// TIA Portal V20 export
DATA_BLOCK "LBP_SentronPac"   // DB1001
TITLE = SENTRON PAC
{ S7_Optimized_Access := 'FALSE'; DB_Accessible_From_OPC_UA := 'FALSE' }
AUTHOR : SINUMERIK
FAMILY : SINUMERIK_ONE
VERSION : 6.24
// Interface between user program and operating software, contains signals for SENTRON PAC energy monitoring devices / Interface entre programme utilisateur et logiciel d'exploitation, contient des signaux pour unités de surveillance de l'énergie SENTRON PAC
// stored: AutoNumber false, DBAccessibleFromOPCUA false, DBAccessibleFromWebserver false
   VAR RETAIN
      ManualVal { ExternalWritable := 'False'} : Bool;   // Display of manual value / Affichage de la valeur manuelle
      SentronPacMach { ExternalWritable := 'False'} : Bool;   // Sentron PAC represented machine / Machine représentée par Sentron PAC
      FeedInEnergyReadSP { ExternalWritable := 'False'} : Bool;   // Feed-in energy read from Sentron PAC / Énergie alimentée mesurée par Sentron PAC
      FeedBackEnergyReadSP { ExternalWritable := 'False'} : Bool;   // Feed back energy read from Sentron PAC / Énergie réinjectée mesurée par Sentron PAC
      FeedInEnergyReadAuxil { ExternalWritable := 'False'} : Bool;   // Feed-in energy read auxiliary / Énergie alimentée, mesurée par AUX
      FeedBackEnergyReadAuxil { ExternalWritable := 'False'} : Bool;   // Feed back energy read auxiliary / Énergie réinjectée, mesurée par AUX
      res0_6 { ExternalWritable := 'False'} : Bool;   // Reserved / Réservé
      res0_7 { ExternalWritable := 'False'} : Bool;   // Reserved / Réservé
      MeasAuto { ExternalWritable := 'False'} : Bool;   // Measurement by PLC basic program / Mesure par programme de base AP
      res1_1 { ExternalWritable := 'False'} : Bool;   // Reserved / Réservé
      res1_2 { ExternalWritable := 'False'} : Bool;   // Reserved / Réservé
      res1_3 { ExternalWritable := 'False'} : Bool;   // Reserved / Réservé
      res1_4 { ExternalWritable := 'False'} : Bool;   // Reserved / Réservé
      res1_5 { ExternalWritable := 'False'} : Bool;   // Reserved / Réservé
      res1_6 { ExternalWritable := 'False'} : Bool;   // Reserved / Réservé
      res1_7 { ExternalWritable := 'False'} : Bool;   // Reserved / Réservé
      MeasAct : Bool;   // HMI -> PLC: Active measurement / IHM->AP : Mesure active
      res2_1 { ExternalWritable := 'False'} : Bool;   // Reserved / Réservé
      res2_2 { ExternalWritable := 'False'} : Bool;   // Reserved / Réservé
      res2_3 { ExternalWritable := 'False'} : Bool;   // Reserved / Réservé
      res2_4 { ExternalWritable := 'False'} : Bool;   // Reserved / Réservé
      res2_5 { ExternalWritable := 'False'} : Bool;   // Reserved / Réservé
      res2_6 { ExternalWritable := 'False'} : Bool;   // Reserved / Réservé
      res2_7 { ExternalWritable := 'False'} : Bool;   // Reserved / Réservé
      EStateOn { ExternalWritable := 'False'} : Bool;   // Energy state on / État énergie activé
      res3_1 { ExternalWritable := 'False'} : Bool;   // Reserved / Réservé
      res3_2 { ExternalWritable := 'False'} : Bool;   // Reserved / Réservé
      res3_3 { ExternalWritable := 'False'} : Bool;   // Reserved / Réservé
      res3_4 { ExternalWritable := 'False'} : Bool;   // Reserved / Réservé
      res3_5 { ExternalWritable := 'False'} : Bool;   // Reserved / Réservé
      res3_6 { ExternalWritable := 'False'} : Bool;   // Reserved / Réservé
      res3_7 { ExternalWritable := 'False'} : Bool;   // Reserved / Réservé
      ManualValue { ExternalWritable := 'False'} : Real;   // Manual value / Valeur manuelle
      ActivePowerItem { ExternalWritable := 'False'} : Real;   // Active power item / Puissance active position
      ActiveEnergyItem { ExternalWritable := 'False'} : Real;   // Active energy item / Énergie active position
      ReactiveEnergyItem { ExternalWritable := 'False'} : Real;   // Reactive energy item / Énergie réactive position
      ActivePowerSentron { ExternalWritable := 'False'} : Real;   // Active power from Sentron / Puissance active par Sentron
      ActiveEnergySentron { ExternalWritable := 'False'} : Real;   // Active energy from Sentron / Énergie active par Sentron
      ReactiveEnergySentron { ExternalWritable := 'False'} : Real;   // Reactive energy from Sentron / Énergie réactive par Sentron
      ActiveEnergyDay { ExternalWritable := 'False'} : Real;   // Active energy day / Énergie active jour
      ReactiveEnergyDay { ExternalWritable := 'False'} : Real;   // Reactive energy day / Énergie réactive jour
      ActiveEnergyPrevDay { ExternalWritable := 'False'} : Real;   // Active energy previous day / Énergie active jour précédent
      ReactiveEnergyPrevDay { ExternalWritable := 'False'} : Real;   // Reactive energy previous day / Énergie réactive jour précédent
      ActiveEnergyMonth { ExternalWritable := 'False'} : Real;   // Active energy month / Énergie active mois
      ReactiveEnergyMonth { ExternalWritable := 'False'} : Real;   // Reactive energy month / Énergie réactive mois
      ActiveEnergyPrevMonth { ExternalWritable := 'False'} : Real;   // Active energy previous month / Énergie active mois précédent
      ReactiveEnergyPrevMonth { ExternalWritable := 'False'} : Real;   // Reactive energy previous month / Énergie réactive mois précédent
      ActiveEnergyYear { ExternalWritable := 'False'} : Real;   // Active energy year / Énergie active année
      ReactiveEnergyYear { ExternalWritable := 'False'} : Real;   // Reactive energy year / Énergie réactive année
      ActiveEnergyPrevYear { ExternalWritable := 'False'} : Real;   // Active energy previous year / Énergie active année précédente
      ReactiveEnergyPrevYear { ExternalWritable := 'False'} : Real;   // Reactive energy previous year / Énergie réactive année précédente
      res80 { ExternalWritable := 'False'} : Byte;   // Reserved / Réservé
      res81 { ExternalWritable := 'False'} : Byte;   // Reserved / Réservé
      res82 { ExternalWritable := 'False'} : Byte;   // Reserved / Réservé
      res83 { ExternalWritable := 'False'} : Byte;   // Reserved / Réservé
      res84 { ExternalWritable := 'False'} : Byte;   // Reserved / Réservé
      res85 { ExternalWritable := 'False'} : Byte;   // Reserved / Réservé
      res86 { ExternalWritable := 'False'} : Byte;   // Reserved / Réservé
      res87 { ExternalWritable := 'False'} : Byte;   // Reserved / Réservé
      res88 { ExternalWritable := 'False'} : Real;   // Reserved / Réservé
      res92 { ExternalWritable := 'False'} : Real;   // Reserved / Réservé
      ProductionAct { ExternalWritable := 'False'} : Byte;
      ErrDBD20_NAN { ExternalWritable := 'False'} : Bool;   // DBD20: invalid (not a number) / DBD20 : non valide (pas un nombre)
      ErrDBD24_NAN { ExternalWritable := 'False'} : Bool;   // DBD24: invalid (not a number) / DBD24 : non valide (pas un nombre)
      ErrDBD28_NAN { ExternalWritable := 'False'} : Bool;   // DBD28: invalid (not a number) / DBD28 : non valide (pas un nombre)
      res97_3 { ExternalWritable := 'False'} : Bool;   // Reserved / Réservé
      res97_4 { ExternalWritable := 'False'} : Bool;   // Reserved / Réservé
      res97_5 { ExternalWritable := 'False'} : Bool;   // Reserved / Réservé
      res97_6 { ExternalWritable := 'False'} : Bool;   // Reserved / Réservé
      res97_7 { ExternalWritable := 'False'} : Bool;   // Reserved / Réservé
      ErrDBD104_NAN { ExternalWritable := 'False'} : Bool;   // DBD104: invalid (not a number) / DBD104 : non valide (pas un nombre)
      ErrDBD144_NAN { ExternalWritable := 'False'} : Bool;   // DBD144: invalid (not a number) / DBD144 : non valide (pas un nombre)
      ErrDBD184_NAN { ExternalWritable := 'False'} : Bool;   // DBD184: invalid (not a number) / DBD184 : non valide (pas un nombre)
      ErrDBD224_NAN { ExternalWritable := 'False'} : Bool;   // DBD224: invalid (not a number) / DBD224 : non valide (pas un nombre)
      ErrDBD264_NAN { ExternalWritable := 'False'} : Bool;   // DBD264: invalid (not a number) / DBD264 : non valide (pas un nombre)
      ErrDBD304_NAN { ExternalWritable := 'False'} : Bool;   // DBD304: invalid (not a number) / DBD304 : non valide (pas un nombre)
      ErrDBD344_NAN { ExternalWritable := 'False'} : Bool;   // DBD344: invalid (not a number) / DBD344 : non valide (pas un nombre)
      ErrDBD384_NAN { ExternalWritable := 'False'} : Bool;   // DBD384: invalid (not a number) / DBD384 : non valide (pas un nombre)
      ErrDBD424_NAN { ExternalWritable := 'False'} : Bool;   // DBD424: invalid (not a number) / DBD424 : non valide (pas un nombre)
      ErrDBD464_NAN { ExternalWritable := 'False'} : Bool;   // DBD464: invalid (not a number) / DBD464 : non valide (pas un nombre)
      res99_2 { ExternalWritable := 'False'} : Bool;   // Reserved / Réservé
      res99_3 { ExternalWritable := 'False'} : Bool;   // Reserved / Réservé
      res99_4 { ExternalWritable := 'False'} : Bool;   // Reserved / Réservé
      res99_5 { ExternalWritable := 'False'} : Bool;   // Reserved / Réservé
      res99_6 { ExternalWritable := 'False'} : Bool;   // Reserved / Réservé
      res99_7 { ExternalWritable := 'False'} : Bool;   // Reserved / Réservé
      CtrlE_AuxDevice { ExternalWritable := 'False'} : Array[1..10] of Struct
         ProcessAux : Bool;   // Auxiliary present and to be processed / AUX présent et prêt au traitement
         ReadEnergy : Bool;   // Actual values are refreshed; bit is auto-reset / Les valeurs réelles sont actualisées ; le bit est réinitialisé automatiquement
         MeasAct : Bool;   // Measurement values are computed / Calcul des valeurs de mesure en cours
         MeasMode : Bool;   // Difference of actual values is stored / La différence des valeurs réelles est enregistrée
         InputMode : Bool;   // INPUT "ActivePowerAux" is energy in kWh / INPUT "ActivePowerAux" représente l'énergie en kWh
         res0_5 : Bool;
         res0_6 : Bool;
         ResetAux : Bool;   // Auxiliary data are deleted / Les données AUX sont supprimées
         res1 : Byte;   // Reserved / Réservé
         res2 : Word;   // Reserved / Réservé
         ActivePowerAux : Real;   // [kW]/[kWh] power/energy of auxiliary, written by customer / [kW]/[kWh] puissance/énergie AUX, renseignée par le client
         ActiveEnAux : Real;   // [kWh] actual value of fed-in-energy / [kWh] valeur réelle de l'énergie consommée
         ReActiveEnAux : Real;   // [kWh] actual value of fed-back energy / [kWh] valeur réelle de l'énergie réinjectée
         ActiveEnAuxMeasON : Real;   // [kWh] value of fed-in-energy at start of measurement / [kWh] valeur réelle de l'énergie consommée au début de la mesure
         ReActiveEnAuxMeasON : Real;   // [kWh] value of fed-back energy at start of measurement / Wh] valeur réelle de l'énergie réinjectée au début de la mesure
         ActiveEnAuxMeasOFF : Real;   // [kWh] value of fed-in-energy at end of measurement / [kWh] valeur réelle de l'énergie consommée à la fin de la mesure
         ReActiveEnAuxMeasOFF : Real;   // [kWh] value of fed-back energy at end of measurement / [kWh] valeur réelle de l'énergie réinjectée à la fin de la mesure
         res32 : DWord;   // Reserved / Réservé
         res36 : Real;   // Reserved / Réservé
      END_STRUCT;
   END_VAR
BEGIN
   // CtrlE_AuxDevice[2].ProcessAux : Auxiliary present and to be processed / AUX présent et prêt au traitement
   // CtrlE_AuxDevice[3].ProcessAux : Auxiliary present and to be processed / AUX présent et prêt au traitement
   // CtrlE_AuxDevice[4].ProcessAux : Auxiliary present and to be processed / AUX présent et prêt au traitement
   // CtrlE_AuxDevice[5].ProcessAux : Auxiliary present and to be processed / AUX présent et prêt au traitement
   // CtrlE_AuxDevice[6].ProcessAux : Auxiliary present and to be processed / AUX présent et prêt au traitement
   // CtrlE_AuxDevice[7].ProcessAux : Auxiliary present and to be processed / AUX présent et prêt au traitement
   // CtrlE_AuxDevice[8].ProcessAux : Auxiliary present and to be processed / AUX présent et prêt au traitement
   // CtrlE_AuxDevice[9].ProcessAux : Auxiliary present and to be processed / AUX présent et prêt au traitement
   // CtrlE_AuxDevice[10].ProcessAux : Auxiliary present and to be processed / AUX présent et prêt au traitement
   // CtrlE_AuxDevice[2].ReadEnergy : Actual values are refreshed; bit is auto-reset / Les valeurs réelles sont actualisées ; le bit est réinitialisé automatiquement
   // CtrlE_AuxDevice[3].ReadEnergy : Actual values are refreshed; bit is auto-reset / Les valeurs réelles sont actualisées ; le bit est réinitialisé automatiquement
   // CtrlE_AuxDevice[4].ReadEnergy : Actual values are refreshed; bit is auto-reset / Les valeurs réelles sont actualisées ; le bit est réinitialisé automatiquement
   // CtrlE_AuxDevice[5].ReadEnergy : Actual values are refreshed; bit is auto-reset / Les valeurs réelles sont actualisées ; le bit est réinitialisé automatiquement
   // CtrlE_AuxDevice[6].ReadEnergy : Actual values are refreshed; bit is auto-reset / Les valeurs réelles sont actualisées ; le bit est réinitialisé automatiquement
   // CtrlE_AuxDevice[7].ReadEnergy : Actual values are refreshed; bit is auto-reset / Les valeurs réelles sont actualisées ; le bit est réinitialisé automatiquement
   // CtrlE_AuxDevice[8].ReadEnergy : Actual values are refreshed; bit is auto-reset / Les valeurs réelles sont actualisées ; le bit est réinitialisé automatiquement
   // CtrlE_AuxDevice[9].ReadEnergy : Actual values are refreshed; bit is auto-reset / Les valeurs réelles sont actualisées ; le bit est réinitialisé automatiquement
   // CtrlE_AuxDevice[10].ReadEnergy : Actual values are refreshed; bit is auto-reset / Les valeurs réelles sont actualisées ; le bit est réinitialisé automatiquement
   // CtrlE_AuxDevice[2].MeasAct : Measurement values are computed / Calcul des valeurs de mesure en cours
   // CtrlE_AuxDevice[3].MeasAct : Measurement values are computed / Calcul des valeurs de mesure en cours
   // CtrlE_AuxDevice[4].MeasAct : Measurement values are computed / Calcul des valeurs de mesure en cours
   // CtrlE_AuxDevice[5].MeasAct : Measurement values are computed / Calcul des valeurs de mesure en cours
   // CtrlE_AuxDevice[6].MeasAct : Measurement values are computed / Calcul des valeurs de mesure en cours
   // CtrlE_AuxDevice[7].MeasAct : Measurement values are computed / Calcul des valeurs de mesure en cours
   // CtrlE_AuxDevice[8].MeasAct : Measurement values are computed / Calcul des valeurs de mesure en cours
   // CtrlE_AuxDevice[9].MeasAct : Measurement values are computed / Calcul des valeurs de mesure en cours
   // CtrlE_AuxDevice[10].MeasAct : Measurement values are computed / Calcul des valeurs de mesure en cours
   // CtrlE_AuxDevice[2].MeasMode : Difference of actual values is stored / La différence des valeurs réelles est enregistrée
   // CtrlE_AuxDevice[3].MeasMode : Difference of actual values is stored / La différence des valeurs réelles est enregistrée
   // CtrlE_AuxDevice[4].MeasMode : Difference of actual values is stored / La différence des valeurs réelles est enregistrée
   // CtrlE_AuxDevice[5].MeasMode : Difference of actual values is stored / La différence des valeurs réelles est enregistrée
   // CtrlE_AuxDevice[6].MeasMode : Difference of actual values is stored / La différence des valeurs réelles est enregistrée
   // CtrlE_AuxDevice[7].MeasMode : Difference of actual values is stored / La différence des valeurs réelles est enregistrée
   // CtrlE_AuxDevice[8].MeasMode : Difference of actual values is stored / La différence des valeurs réelles est enregistrée
   // CtrlE_AuxDevice[9].MeasMode : Difference of actual values is stored / La différence des valeurs réelles est enregistrée
   // CtrlE_AuxDevice[10].MeasMode : Difference of actual values is stored / La différence des valeurs réelles est enregistrée
   // CtrlE_AuxDevice[2].InputMode : INPUT "ActivePowerAux" is energy in kWh / INPUT "ActivePowerAux" représente l'énergie en kWh
   // CtrlE_AuxDevice[3].InputMode : INPUT "ActivePowerAux" is energy in kWh / INPUT "ActivePowerAux" représente l'énergie en kWh
   // CtrlE_AuxDevice[4].InputMode : INPUT "ActivePowerAux" is energy in kWh / INPUT "ActivePowerAux" représente l'énergie en kWh
   // CtrlE_AuxDevice[5].InputMode : INPUT "ActivePowerAux" is energy in kWh / INPUT "ActivePowerAux" représente l'énergie en kWh
   // CtrlE_AuxDevice[6].InputMode : INPUT "ActivePowerAux" is energy in kWh / INPUT "ActivePowerAux" représente l'énergie en kWh
   // CtrlE_AuxDevice[7].InputMode : INPUT "ActivePowerAux" is energy in kWh / INPUT "ActivePowerAux" représente l'énergie en kWh
   // CtrlE_AuxDevice[8].InputMode : INPUT "ActivePowerAux" is energy in kWh / INPUT "ActivePowerAux" représente l'énergie en kWh
   // CtrlE_AuxDevice[9].InputMode : INPUT "ActivePowerAux" is energy in kWh / INPUT "ActivePowerAux" représente l'énergie en kWh
   // CtrlE_AuxDevice[10].InputMode : INPUT "ActivePowerAux" is energy in kWh / INPUT "ActivePowerAux" représente l'énergie en kWh
   // CtrlE_AuxDevice[2].ResetAux : Auxiliary data are deleted / Les données AUX sont supprimées
   // CtrlE_AuxDevice[3].ResetAux : Auxiliary data are deleted / Les données AUX sont supprimées
   // CtrlE_AuxDevice[4].ResetAux : Auxiliary data are deleted / Les données AUX sont supprimées
   // CtrlE_AuxDevice[5].ResetAux : Auxiliary data are deleted / Les données AUX sont supprimées
   // CtrlE_AuxDevice[6].ResetAux : Auxiliary data are deleted / Les données AUX sont supprimées
   // CtrlE_AuxDevice[7].ResetAux : Auxiliary data are deleted / Les données AUX sont supprimées
   // CtrlE_AuxDevice[8].ResetAux : Auxiliary data are deleted / Les données AUX sont supprimées
   // CtrlE_AuxDevice[9].ResetAux : Auxiliary data are deleted / Les données AUX sont supprimées
   // CtrlE_AuxDevice[10].ResetAux : Auxiliary data are deleted / Les données AUX sont supprimées
   // CtrlE_AuxDevice[2].res1 : Reserved / Réservé
   // CtrlE_AuxDevice[3].res1 : Reserved / Réservé
   // CtrlE_AuxDevice[4].res1 : Reserved / Réservé
   // CtrlE_AuxDevice[5].res1 : Reserved / Réservé
   // CtrlE_AuxDevice[6].res1 : Reserved / Réservé
   // CtrlE_AuxDevice[7].res1 : Reserved / Réservé
   // CtrlE_AuxDevice[8].res1 : Reserved / Réservé
   // CtrlE_AuxDevice[9].res1 : Reserved / Réservé
   // CtrlE_AuxDevice[10].res1 : Reserved / Réservé
   // CtrlE_AuxDevice[2].res2 : Reserved / Réservé
   // CtrlE_AuxDevice[3].res2 : Reserved / Réservé
   // CtrlE_AuxDevice[4].res2 : Reserved / Réservé
   // CtrlE_AuxDevice[5].res2 : Reserved / Réservé
   // CtrlE_AuxDevice[6].res2 : Reserved / Réservé
   // CtrlE_AuxDevice[7].res2 : Reserved / Réservé
   // CtrlE_AuxDevice[8].res2 : Reserved / Réservé
   // CtrlE_AuxDevice[9].res2 : Reserved / Réservé
   // CtrlE_AuxDevice[10].res2 : Reserved / Réservé
   // CtrlE_AuxDevice[2].ActivePowerAux : [kW]/[kWh] power/energy of auxiliary, written by customer / [kW]/[kWh] puissance/énergie AUX, renseignée par le client
   // CtrlE_AuxDevice[3].ActivePowerAux : [kW]/[kWh] power/energy of auxiliary, written by customer / [kW]/[kWh] puissance/énergie AUX, renseignée par le client
   // CtrlE_AuxDevice[4].ActivePowerAux : [kW]/[kWh] power/energy of auxiliary, written by customer / [kW]/[kWh] puissance/énergie AUX, renseignée par le client
   // CtrlE_AuxDevice[5].ActivePowerAux : [kW]/[kWh] power/energy of auxiliary, written by customer / [kW]/[kWh] puissance/énergie AUX, renseignée par le client
   // CtrlE_AuxDevice[6].ActivePowerAux : [kW]/[kWh] power/energy of auxiliary, written by customer / [kW]/[kWh] puissance/énergie AUX, renseignée par le client
   // CtrlE_AuxDevice[7].ActivePowerAux : [kW]/[kWh] power/energy of auxiliary, written by customer / [kW]/[kWh] puissance/énergie AUX, renseignée par le client
   // CtrlE_AuxDevice[8].ActivePowerAux : [kW]/[kWh] power/energy of auxiliary, written by customer / [kW]/[kWh] puissance/énergie AUX, renseignée par le client
   // CtrlE_AuxDevice[9].ActivePowerAux : [kW]/[kWh] power/energy of auxiliary, written by customer / [kW]/[kWh] puissance/énergie AUX, renseignée par le client
   // CtrlE_AuxDevice[10].ActivePowerAux : [kW]/[kWh] power/energy of auxiliary, written by customer / [kW]/[kWh] puissance/énergie AUX, renseignée par le client
   // CtrlE_AuxDevice[2].ActiveEnAux : [kWh] actual value of fed-in-energy / [kWh] valeur réelle de l'énergie consommée
   // CtrlE_AuxDevice[3].ActiveEnAux : [kWh] actual value of fed-in-energy / [kWh] valeur réelle de l'énergie consommée
   // CtrlE_AuxDevice[4].ActiveEnAux : [kWh] actual value of fed-in-energy / [kWh] valeur réelle de l'énergie consommée
   // CtrlE_AuxDevice[5].ActiveEnAux : [kWh] actual value of fed-in-energy / [kWh] valeur réelle de l'énergie consommée
   // CtrlE_AuxDevice[6].ActiveEnAux : [kWh] actual value of fed-in-energy / [kWh] valeur réelle de l'énergie consommée
   // CtrlE_AuxDevice[7].ActiveEnAux : [kWh] actual value of fed-in-energy / [kWh] valeur réelle de l'énergie consommée
   // CtrlE_AuxDevice[8].ActiveEnAux : [kWh] actual value of fed-in-energy / [kWh] valeur réelle de l'énergie consommée
   // CtrlE_AuxDevice[9].ActiveEnAux : [kWh] actual value of fed-in-energy / [kWh] valeur réelle de l'énergie consommée
   // CtrlE_AuxDevice[10].ActiveEnAux : [kWh] actual value of fed-in-energy / [kWh] valeur réelle de l'énergie consommée
   // CtrlE_AuxDevice[2].ReActiveEnAux : [kWh] actual value of fed-back energy / [kWh] valeur réelle de l'énergie réinjectée
   // CtrlE_AuxDevice[3].ReActiveEnAux : [kWh] actual value of fed-back energy / [kWh] valeur réelle de l'énergie réinjectée
   // CtrlE_AuxDevice[4].ReActiveEnAux : [kWh] actual value of fed-back energy / [kWh] valeur réelle de l'énergie réinjectée
   // CtrlE_AuxDevice[5].ReActiveEnAux : [kWh] actual value of fed-back energy / [kWh] valeur réelle de l'énergie réinjectée
   // CtrlE_AuxDevice[6].ReActiveEnAux : [kWh] actual value of fed-back energy / [kWh] valeur réelle de l'énergie réinjectée
   // CtrlE_AuxDevice[7].ReActiveEnAux : [kWh] actual value of fed-back energy / [kWh] valeur réelle de l'énergie réinjectée
   // CtrlE_AuxDevice[8].ReActiveEnAux : [kWh] actual value of fed-back energy / [kWh] valeur réelle de l'énergie réinjectée
   // CtrlE_AuxDevice[9].ReActiveEnAux : [kWh] actual value of fed-back energy / [kWh] valeur réelle de l'énergie réinjectée
   // CtrlE_AuxDevice[10].ReActiveEnAux : [kWh] actual value of fed-back energy / [kWh] valeur réelle de l'énergie réinjectée
   // CtrlE_AuxDevice[2].ActiveEnAuxMeasON : [kWh] value of fed-in-energy at start of measurement / [kWh] valeur réelle de l'énergie consommée au début de la mesure
   // CtrlE_AuxDevice[3].ActiveEnAuxMeasON : [kWh] value of fed-in-energy at start of measurement / [kWh] valeur réelle de l'énergie consommée au début de la mesure
   // CtrlE_AuxDevice[4].ActiveEnAuxMeasON : [kWh] value of fed-in-energy at start of measurement / [kWh] valeur réelle de l'énergie consommée au début de la mesure
   // CtrlE_AuxDevice[5].ActiveEnAuxMeasON : [kWh] value of fed-in-energy at start of measurement / [kWh] valeur réelle de l'énergie consommée au début de la mesure
   // CtrlE_AuxDevice[6].ActiveEnAuxMeasON : [kWh] value of fed-in-energy at start of measurement / [kWh] valeur réelle de l'énergie consommée au début de la mesure
   // CtrlE_AuxDevice[7].ActiveEnAuxMeasON : [kWh] value of fed-in-energy at start of measurement / [kWh] valeur réelle de l'énergie consommée au début de la mesure
   // CtrlE_AuxDevice[8].ActiveEnAuxMeasON : [kWh] value of fed-in-energy at start of measurement / [kWh] valeur réelle de l'énergie consommée au début de la mesure
   // CtrlE_AuxDevice[9].ActiveEnAuxMeasON : [kWh] value of fed-in-energy at start of measurement / [kWh] valeur réelle de l'énergie consommée au début de la mesure
   // CtrlE_AuxDevice[10].ActiveEnAuxMeasON : [kWh] value of fed-in-energy at start of measurement / [kWh] valeur réelle de l'énergie consommée au début de la mesure
   // CtrlE_AuxDevice[2].ReActiveEnAuxMeasON : [kWh] value of fed-back energy at start of measurement / Wh] valeur réelle de l'énergie réinjectée au début de la mesure
   // CtrlE_AuxDevice[3].ReActiveEnAuxMeasON : [kWh] value of fed-back energy at start of measurement / Wh] valeur réelle de l'énergie réinjectée au début de la mesure
   // CtrlE_AuxDevice[4].ReActiveEnAuxMeasON : [kWh] value of fed-back energy at start of measurement / Wh] valeur réelle de l'énergie réinjectée au début de la mesure
   // CtrlE_AuxDevice[5].ReActiveEnAuxMeasON : [kWh] value of fed-back energy at start of measurement / Wh] valeur réelle de l'énergie réinjectée au début de la mesure
   // CtrlE_AuxDevice[6].ReActiveEnAuxMeasON : [kWh] value of fed-back energy at start of measurement / Wh] valeur réelle de l'énergie réinjectée au début de la mesure
   // CtrlE_AuxDevice[7].ReActiveEnAuxMeasON : [kWh] value of fed-back energy at start of measurement / Wh] valeur réelle de l'énergie réinjectée au début de la mesure
   // CtrlE_AuxDevice[8].ReActiveEnAuxMeasON : [kWh] value of fed-back energy at start of measurement / Wh] valeur réelle de l'énergie réinjectée au début de la mesure
   // CtrlE_AuxDevice[9].ReActiveEnAuxMeasON : [kWh] value of fed-back energy at start of measurement / Wh] valeur réelle de l'énergie réinjectée au début de la mesure
   // CtrlE_AuxDevice[10].ReActiveEnAuxMeasON : [kWh] value of fed-back energy at start of measurement / Wh] valeur réelle de l'énergie réinjectée au début de la mesure
   // CtrlE_AuxDevice[2].ActiveEnAuxMeasOFF : [kWh] value of fed-in-energy at end of measurement / [kWh] valeur réelle de l'énergie consommée à la fin de la mesure
   // CtrlE_AuxDevice[3].ActiveEnAuxMeasOFF : [kWh] value of fed-in-energy at end of measurement / [kWh] valeur réelle de l'énergie consommée à la fin de la mesure
   // CtrlE_AuxDevice[4].ActiveEnAuxMeasOFF : [kWh] value of fed-in-energy at end of measurement / [kWh] valeur réelle de l'énergie consommée à la fin de la mesure
   // CtrlE_AuxDevice[5].ActiveEnAuxMeasOFF : [kWh] value of fed-in-energy at end of measurement / [kWh] valeur réelle de l'énergie consommée à la fin de la mesure
   // CtrlE_AuxDevice[6].ActiveEnAuxMeasOFF : [kWh] value of fed-in-energy at end of measurement / [kWh] valeur réelle de l'énergie consommée à la fin de la mesure
   // CtrlE_AuxDevice[7].ActiveEnAuxMeasOFF : [kWh] value of fed-in-energy at end of measurement / [kWh] valeur réelle de l'énergie consommée à la fin de la mesure
   // CtrlE_AuxDevice[8].ActiveEnAuxMeasOFF : [kWh] value of fed-in-energy at end of measurement / [kWh] valeur réelle de l'énergie consommée à la fin de la mesure
   // CtrlE_AuxDevice[9].ActiveEnAuxMeasOFF : [kWh] value of fed-in-energy at end of measurement / [kWh] valeur réelle de l'énergie consommée à la fin de la mesure
   // CtrlE_AuxDevice[10].ActiveEnAuxMeasOFF : [kWh] value of fed-in-energy at end of measurement / [kWh] valeur réelle de l'énergie consommée à la fin de la mesure
   // CtrlE_AuxDevice[2].ReActiveEnAuxMeasOFF : [kWh] value of fed-back energy at end of measurement / [kWh] valeur réelle de l'énergie réinjectée à la fin de la mesure
   // CtrlE_AuxDevice[3].ReActiveEnAuxMeasOFF : [kWh] value of fed-back energy at end of measurement / [kWh] valeur réelle de l'énergie réinjectée à la fin de la mesure
   // CtrlE_AuxDevice[4].ReActiveEnAuxMeasOFF : [kWh] value of fed-back energy at end of measurement / [kWh] valeur réelle de l'énergie réinjectée à la fin de la mesure
   // CtrlE_AuxDevice[5].ReActiveEnAuxMeasOFF : [kWh] value of fed-back energy at end of measurement / [kWh] valeur réelle de l'énergie réinjectée à la fin de la mesure
   // CtrlE_AuxDevice[6].ReActiveEnAuxMeasOFF : [kWh] value of fed-back energy at end of measurement / [kWh] valeur réelle de l'énergie réinjectée à la fin de la mesure
   // CtrlE_AuxDevice[7].ReActiveEnAuxMeasOFF : [kWh] value of fed-back energy at end of measurement / [kWh] valeur réelle de l'énergie réinjectée à la fin de la mesure
   // CtrlE_AuxDevice[8].ReActiveEnAuxMeasOFF : [kWh] value of fed-back energy at end of measurement / [kWh] valeur réelle de l'énergie réinjectée à la fin de la mesure
   // CtrlE_AuxDevice[9].ReActiveEnAuxMeasOFF : [kWh] value of fed-back energy at end of measurement / [kWh] valeur réelle de l'énergie réinjectée à la fin de la mesure
   // CtrlE_AuxDevice[10].ReActiveEnAuxMeasOFF : [kWh] value of fed-back energy at end of measurement / [kWh] valeur réelle de l'énergie réinjectée à la fin de la mesure
   // CtrlE_AuxDevice[2].res32 : Reserved / Réservé
   // CtrlE_AuxDevice[3].res32 : Reserved / Réservé
   // CtrlE_AuxDevice[4].res32 : Reserved / Réservé
   // CtrlE_AuxDevice[5].res32 : Reserved / Réservé
   // CtrlE_AuxDevice[6].res32 : Reserved / Réservé
   // CtrlE_AuxDevice[7].res32 : Reserved / Réservé
   // CtrlE_AuxDevice[8].res32 : Reserved / Réservé
   // CtrlE_AuxDevice[9].res32 : Reserved / Réservé
   // CtrlE_AuxDevice[10].res32 : Reserved / Réservé
   // CtrlE_AuxDevice[2].res36 : Reserved / Réservé
   // CtrlE_AuxDevice[3].res36 : Reserved / Réservé
   // CtrlE_AuxDevice[4].res36 : Reserved / Réservé
   // CtrlE_AuxDevice[5].res36 : Reserved / Réservé
   // CtrlE_AuxDevice[6].res36 : Reserved / Réservé
   // CtrlE_AuxDevice[7].res36 : Reserved / Réservé
   // CtrlE_AuxDevice[8].res36 : Reserved / Réservé
   // CtrlE_AuxDevice[9].res36 : Reserved / Réservé
   // CtrlE_AuxDevice[10].res36 : Reserved / Réservé
END_DATA_BLOCK
